INTERFACE I_LINT EXTENDS I_Datatype

{warning disable C5410}
PROPERTY PUBLIC Value : REFERENCE TO LINT
{warning restore C5410}
GET
END_GET
END_PROPERTY

END_INTERFACE

(* stored: Version 1.1.0.1, ProductVersion 3.1.4024.15
   Itf I_LINT: Id {4e7d2ae8-e548-0bb8-2964-4fb72c9e560b}
   Property Value: Id {3b53851b-99be-05f4-28ef-d7a8d0e41384}
   Get Get: Id {697c86f9-c94b-05e3-23c0-d3d99e317c39} *)
